FUNCTION_BLOCK ResetValvesManager (* Composite Function Block Type *)
  (* Standard: 61499-2 *)
  (* Version 0.0, 8/20/2024, SESA713705, Schneider Electric, template *)
  PACKAGE SE.Nereda;
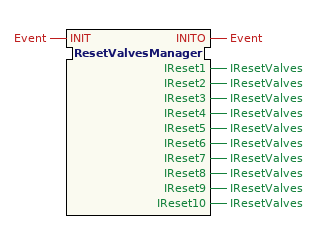
  EVENT_INPUT
    INIT;
  END_EVENT
  EVENT_OUTPUT
    INITO;
  END_EVENT
  PLUGS
    IReset1 : IResetValves;
    IReset2 : IResetValves;
    IReset3 : IResetValves;
    IReset4 : IResetValves;
    IReset5 : IResetValves;
    IReset6 : IResetValves;
    IReset7 : IResetValves;
    IReset8 : IResetValves;
    IReset9 : IResetValves;
    IReset10 : IResetValves;
  END_PLUGS
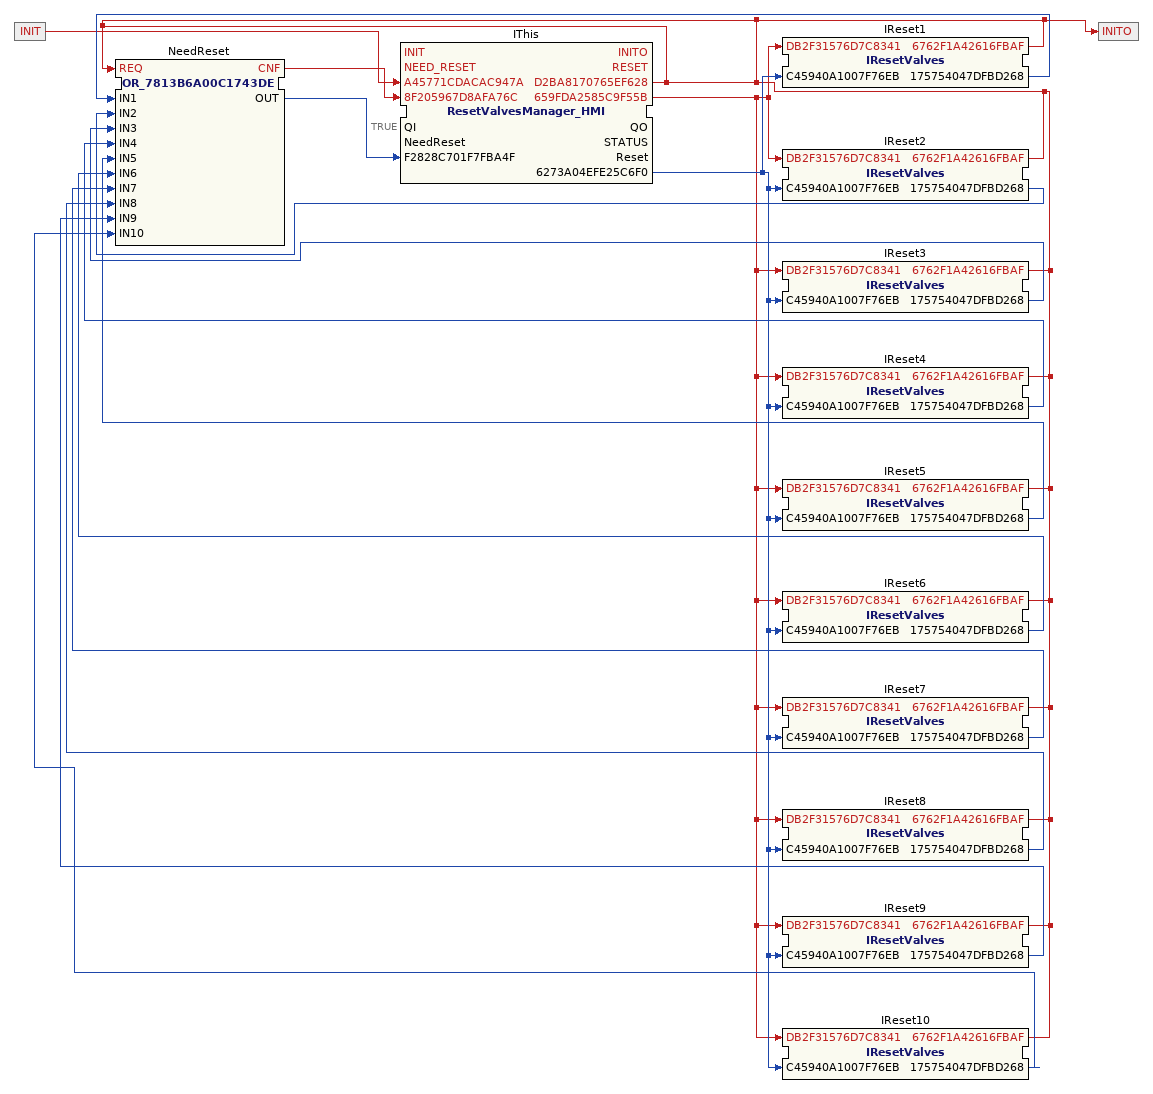
  FBS
    IThis : ResetValvesManager_HMI(QI := TRUE);
    NeedReset : OR_7813B6A00C1743DE; {SET_ATTRIBUTE(Configuration.GenericFBType.InterfaceParams, Runtime.Standard#CNT:=10;OUT:BOOL)}
  END_FBS
  EVENT_CONNECTIONS
    IReset1.6762F1A42616FBAF TO NeedReset.REQ;
    IReset2.6762F1A42616FBAF TO NeedReset.REQ;
    IReset3.6762F1A42616FBAF TO NeedReset.REQ;
    IReset4.6762F1A42616FBAF TO NeedReset.REQ;
    IReset5.6762F1A42616FBAF TO NeedReset.REQ;
    IReset6.6762F1A42616FBAF TO NeedReset.REQ;
    IReset7.6762F1A42616FBAF TO NeedReset.REQ;
    IReset8.6762F1A42616FBAF TO NeedReset.REQ;
    IReset9.6762F1A42616FBAF TO NeedReset.REQ;
    IReset10.6762F1A42616FBAF TO NeedReset.REQ;
    INIT TO IThis.A45771CDACAC947A;
    NeedReset.CNF TO IThis.8F205967D8AFA76C;
    IThis.D2BA8170765EF628 TO INITO;
    IThis.D2BA8170765EF628 TO NeedReset.REQ;
    IThis.659FDA2585C9F55B TO IReset1.DB2F31576D7C8341;
    IThis.659FDA2585C9F55B TO IReset2.DB2F31576D7C8341;
    IThis.659FDA2585C9F55B TO IReset3.DB2F31576D7C8341;
    IThis.659FDA2585C9F55B TO IReset4.DB2F31576D7C8341;
    IThis.659FDA2585C9F55B TO IReset5.DB2F31576D7C8341;
    IThis.659FDA2585C9F55B TO IReset6.DB2F31576D7C8341;
    IThis.659FDA2585C9F55B TO IReset7.DB2F31576D7C8341;
    IThis.659FDA2585C9F55B TO IReset8.DB2F31576D7C8341;
    IThis.659FDA2585C9F55B TO IReset9.DB2F31576D7C8341;
    IThis.659FDA2585C9F55B TO IReset10.DB2F31576D7C8341;
  END_CONNECTIONS
  DATA_CONNECTIONS
    IReset1.175754047DFBD268 TO NeedReset.IN1;
    IReset2.175754047DFBD268 TO NeedReset.IN2;
    NeedReset.OUT TO IThis.F2828C701F7FBA4F;
    IThis.6273A04EFE25C6F0 TO IReset1.C45940A1007F76EB;
    IThis.6273A04EFE25C6F0 TO IReset2.C45940A1007F76EB;
    IThis.6273A04EFE25C6F0 TO IReset3.C45940A1007F76EB;
    IThis.6273A04EFE25C6F0 TO IReset4.C45940A1007F76EB;
    IThis.6273A04EFE25C6F0 TO IReset5.C45940A1007F76EB;
    IThis.6273A04EFE25C6F0 TO IReset6.C45940A1007F76EB;
    IThis.6273A04EFE25C6F0 TO IReset7.C45940A1007F76EB;
    IThis.6273A04EFE25C6F0 TO IReset8.C45940A1007F76EB;
    IThis.6273A04EFE25C6F0 TO IReset9.C45940A1007F76EB;
    IThis.6273A04EFE25C6F0 TO IReset10.C45940A1007F76EB;
    IReset3.175754047DFBD268 TO NeedReset.IN3;
    IReset4.175754047DFBD268 TO NeedReset.IN4;
    IReset5.175754047DFBD268 TO NeedReset.IN5;
    IReset6.175754047DFBD268 TO NeedReset.IN6;
    IReset7.175754047DFBD268 TO NeedReset.IN7;
    IReset8.175754047DFBD268 TO NeedReset.IN8;
    IReset9.175754047DFBD268 TO NeedReset.IN9;
    IReset10.175754047DFBD268 TO NeedReset.IN10;
  END_CONNECTIONS
END_FUNCTION_BLOCK
